FUNCTION_BLOCK ControlPanel
VAR_INPUT
END_VAR
VAR_OUTPUT
END_VAR
VAR
	bAtBufferEntry	:	BOOL;
	
	
END_VAR

{region "READ Values from Sensors"}
	bAtBufferEntry	:=	GVL.mb_Output_Coils[0];
		 
		 
{endregion}

END_FUNCTION_BLOCK

(* stored: Version 1.1.0.1, ProductVersion 3.1.4024.12
   POU ControlPanel: Id {6fafcdca-fd53-44b1-8233-794b801bcaa5}, SpecialFunc None *)
